PROGRAM MAIN
VAR
END_VAR

END_PROGRAM

(* stored: Version 1.1.0.1
   POU MAIN: Id {4d23361e-5531-43ee-8b6f-df7299a7184c} *)
